{attribute 'qualified_only'}
{attribute 'strict'}
TYPE E_Controlmode :
(
	IO_Testmode		:= 0,
	Manual			:= 1,
	Test_individual	:= 2,
	Test_sequence	:= 3	
) BYTE;
END_TYPE

(* stored: Version 1.1.0.1, ProductVersion 3.1.4024.11
   DUT E_Controlmode: Id {65fb7a46-c119-4bd1-bf4a-52872c444a42} *)
